FUNCTION_BLOCK basicBloqueioAtivaDesativa (* Basic Function Block Type *)
  (* Standard: 61499-2 *)
  (* Version 0.0, 02/03/2026, Template *)
  PACKAGE Hidryco.HidrycoLib;
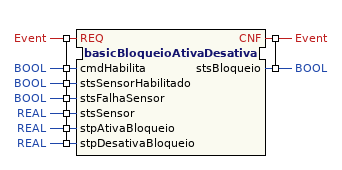
  EVENT_INPUT
    REQ WITH cmdHabilita, stsSensorHabilitado, stsFalhaSensor, stsSensor, stpAtivaBloqueio, stpDesativaBloqueio;
  END_EVENT
  EVENT_OUTPUT
    CNF WITH stsBloqueio;
  END_EVENT
  VAR_INPUT
    cmdHabilita : BOOL;
    stsSensorHabilitado : BOOL;
    stsFalhaSensor : BOOL;
    stsSensor : REAL;
    stpAtivaBloqueio : REAL;
    stpDesativaBloqueio : REAL;
  END_VAR
  VAR_OUTPUT
    stsBloqueio : BOOL;
  END_VAR
  VAR
    bBloqueioNivel : BOOL;
    bBloqueioAnt : BOOL;
    bMudou : BOOL;
  END_VAR
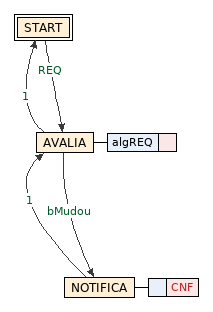
  EC_STATES
    START; (* Initial State *)
    AVALIA : algREQ;
    NOTIFICA : -> CNF;
  END_STATES
  EC_TRANSITIONS
    START TO AVALIA := REQ;
    AVALIA TO NOTIFICA := bMudou;
    AVALIA TO START := 1;
    NOTIFICA TO AVALIA := 1;
  END_TRANSITIONS
  ALGORITHM algREQ IN ST:
bBloqueioAnt := stsBloqueio;

IF NOT cmdHabilita THEN
    (* bloqueio desabilitado *)
    stsBloqueio := FALSE;

ELSIF NOT stsSensorHabilitado OR stsFalhaSensor THEN
    (* sensor indisponível *)
    stsBloqueio := TRUE;

ELSIF stpAtivaBloqueio = stpDesativaBloqueio THEN
    (* setpoints iguais: configuração inválida *)
    stsBloqueio := TRUE;

ELSIF stpAtivaBloqueio < stpDesativaBloqueio THEN
    (* nível baixo *)
    IF stsSensor < stpAtivaBloqueio THEN
        bBloqueioNivel := TRUE;
    ELSIF stsSensor >= stpDesativaBloqueio THEN
        bBloqueioNivel := FALSE;
    END_IF;
    stsBloqueio := bBloqueioNivel;

ELSE
    (* nível alto *)
    IF stsSensor > stpAtivaBloqueio THEN
        bBloqueioNivel := TRUE;
    ELSIF stsSensor <= stpDesativaBloqueio THEN
        bBloqueioNivel := FALSE;
    END_IF;
    stsBloqueio := bBloqueioNivel;
END_IF;

bMudou := (stsBloqueio <> bBloqueioAnt);
;
  END_ALGORITHM
END_FUNCTION_BLOCK
